// TIA Portal V20 export
// export: Created 2025-12-01T14:57:27.5166691Z, ExportSetting None, DisplayName Totally Integrated Automation Portal, DisplayVersion V20 Update 3, DisplayName TIA Portal Openness, DisplayVersion V20 Update 3, DisplayName TIA Portal Version Control Interface, DisplayVersion V20 Update 3, DisplayName STEP 7 Professional, DisplayVersion V20 Update 3, DisplayName STEP 7 Safety, DisplayVersion V20 Update 2, DisplayName WinCC Basic/Comfort/Advanced, DisplayVersion V20 Update 3, DisplayName WinCC Professional, DisplayVersion V20 Update 3, DisplayName WinCC Unified, DisplayVersion V20 Update 3
FUNCTION_BLOCK "FB606_SalidaMovil_Lateral_EnDesCarga_Quimarox"   // FB606, LAD
{ S7_Optimized_Access := 'FALSE' }
// stored: AutoNumber false, SetENOAutomatically false
   VAR_INPUT
      MesaSiguiente : UInt;
      MesaDeDescarga : UInt;
      ID_Quimarox : UInt;
      ID_Elemento : UInt;
      DestinoAsociado : UInt;
      EnTension : Bool;
      Termico : Bool;
      pHs_PosicionDescarga : Bool;
      pHs_Protrusion : Bool;
      En_PosicionDescarga : Bool;
      En_PosicionReposo : Bool;
      NXT_PTF : Bool;
      NXT_FTF : Bool;
      V_FILTRO_pHsPresencia : Int;
      Pto_Ajuste_1 : Int;   // en mm (paso a lenta en posicionamiento a descarga de transportador)
      Pto_Ajuste_2 : Int;   // en mm (timeout movimiento posicion descarga del transportador)
      Pto_Ajuste_3 : Int;   // en mm (paso a lenta en el proceso de descarga del peine)
      Pto_Ajuste_4 : Int;   // en mm (error protusion en descarga del elevador)
      Pto_Ajuste_5 : Int;   // en mm (paso a lenta en posicionamiento reposo del transportador)
      Pto_Ajuste_6 : Int;   // en mm (timeout movimiento posicion reposo del transportador)
   END_VAR
   VAR_OUTPUT
      NXT_DescargaActiva : Bool;
      NXT_AVTF : Bool;
      ElevadorEnLenta : Bool;
      PararElevador : Bool;
      Avance_SalidaMovil : Bool;
      Ir_PosicionReposo : Bool;
      Ir_PosicionDescarga : Bool;
   END_VAR
   VAR
      TMP_EnTension { S7_SetPoint := 'True'} : "FB910_CNT_UHS";
      FILTRO_pHsPresencia { S7_SetPoint := 'True'} : "FB910_CNT_UHS";
      EstadoAsociadoEnMesa : UInt;
      Ultimo_PeineTratado : UInt;
      Aux_PeineEnDesCarga { ExternalAccessible := 'False'; ExternalVisible := 'False'; ExternalWritable := 'False'} : UInt;
      Siguiente_ParaNosotros : Bool;
      PresenciaEnReset : Bool;
   END_VAR
   VAR_TEMP
      MesaQuimarox : UInt;
      NumeroUT : UInt;
      VagonSiguiente : UInt;
      EsMesaTL : Bool;
      FILTRO_PosicionDesCarga : Bool;
   END_VAR
BEGIN

NETWORK
TITLE = ERROR - Rearme
/////////////////////////////////////////////////////////////
/////////////////////////////////////////////////////////////
/////////////////////////////////////////////////////////////
// Rearne de Errores
      SET;
      A     "DB902_Estado_ZonaMesa".EstadoMesas[#MesaDeDescarga].Rearme_CBx;
      O     "DB902_Estado_ZonaMesa".EstadoMesas[#MesaDeDescarga].PerReset_CBx;
      R     "DB900_Estado_Mesas".EstadoVI[#MesaDeDescarga].Error_Mx;
      R     "DB900_Estado_Mesas".EstadoVI[#MesaDeDescarga].Err_Protusion;
      R     "DB900_Estado_Mesas".EstadoVI[#MesaDeDescarga].Err_Tout_Sacar;
      R     "DB900_Estado_Mesas".EstadoVI[#MesaDeDescarga].Err_Tout_Recoger;
      R     "DB900_Estado_Mesas".EstadoVI[#MesaDeDescarga].Err_DatosPLC;
      R     "DB900_Estado_Mesas".EstadoVI[#MesaDeDescarga].Err_Termico_E1_E3;
      R     "DB900_Estado_Mesas".EstadoVI[#MesaDeDescarga].Err_Perdida_PHs;



NETWORK
TITLE = RECEP OK DE LA ORDEN -- NO SE UTILIZA
/////////////////////////////////////////////////////////////
/////////////////////////////////////////////////////////////
/////////////////////////////////////////////////////////////
// RECEP OK DE LA ORDEN
      SET;
      AN    "DB841_Recepcion".Mesa[#MesaDeDescarga].Protocolo.Ord_S00;
      AN    "DB841_Recepcion".Mesa[#MesaDeDescarga].Protocolo.Ord_S01;
      AN    "DB841_Recepcion".Mesa[#MesaDeDescarga].Protocolo.Ord_S02;
      AN    "DB841_Recepcion".Mesa[#MesaDeDescarga].Protocolo.Ord_S03;
      NOT;
      =     "DB840_Emision".Mesa[#MesaDeDescarga].Protocolo.RecepOK;



NETWORK
TITLE = HMI - Manual
/////////////////////////////////////////////////////////////
/////////////////////////////////////////////////////////////
/////////////////////////////////////////////////////////////
// Para HMI >>> Manual
      SET;
      O     "DB902_Estado_ZonaMesa".EstadoMesas[#MesaDeDescarga].Manual_CBx;
      =     "DB900_Estado_Mesas".EstadoVI[#MesaDeDescarga].Manual;



NETWORK
TITLE = HMI - Entradas y Salidas de la Mesa
/////////////////////////////////////////////////////////////
/////////////////////////////////////////////////////////////
/////////////////////////////////////////////////////////////
// Entradas
      SET;
      A     #pHs_PosicionDescarga;
      =     "DB900_Estado_Mesas".EstadoVI[#MesaDeDescarga].En_PHS_1;
      SET;
      A     #pHs_Protrusion;
      =     "DB900_Estado_Mesas".EstadoVI[#MesaDeDescarga].En_pHs_Prot1;

      SET;
      A     #Termico;
      =     "DB900_Estado_Mesas".EstadoVI[#MesaDeDescarga].En_Termico1;


// Salidas
      SET;
      A     #Avance_SalidaMovil;
      =     "DB900_Estado_Mesas".EstadoVI[#MesaDeDescarga].Sa_Rod_Avance;
      SET;
      A     #Ir_PosicionReposo;
      =     "DB900_Estado_Mesas".EstadoVI[#MesaDeDescarga].Sa_Trans_Baj;
      SET;
      A     #Ir_PosicionDescarga;
      =     "DB900_Estado_Mesas".EstadoVI[#MesaDeDescarga].Sa_Trans_Sub;



NETWORK
TITLE = Comprobacion de que la MESA es de TRACKING
/////////////////////////////////////////////////////////////////////////////////////
/////////////////////////////////////////////////////////////////////////////////////
/////////////////////////////////////////////////////////////////////////////////////
// Comprobar si es una Mesa de Tracking o Routing
      SET;
      A     "DB850_DefinicionMesas".Mesa[#MesaDeDescarga].ConfigMesa.MesaTL;
      =     #EsMesaTL;



REGION Network 6: TMP - Espera En Tension
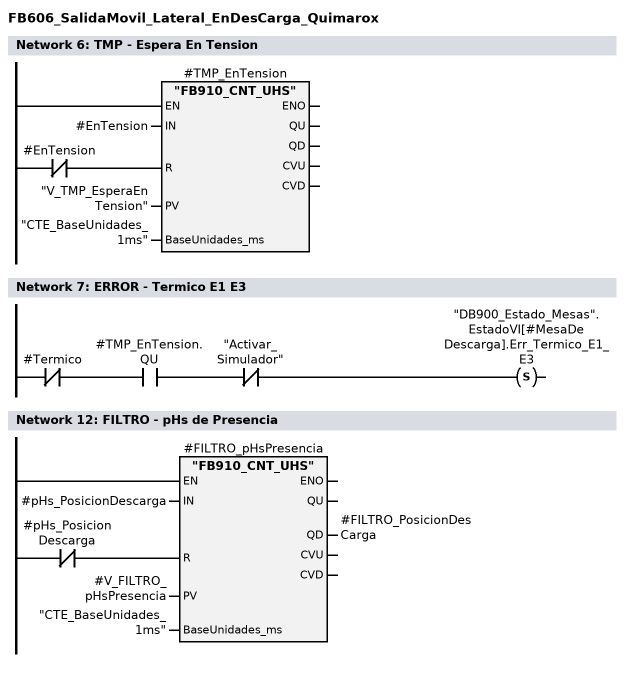
   RUNG wire#powerrail
      #TMP_EnTension(R := wire#w1, IN := #EnTension, PV := "V_TMP_EsperaEnTension", BaseUnidades_ms := "CTE_BaseUnidades_1ms", QU =>, QD =>, CVU =>, CVD =>)
   END_RUNG
   RUNG wire#powerrail
      I_Contact( #EnTension )
   END_RUNG wire#w1
   // the same network as SCL:
   #TMP_EnTension(IN := #EnTension,   // "FB910_CNT_UHS"
                  R := NOT #EnTension,
                  PV := "V_TMP_EsperaEnTension",
                  BaseUnidades_ms := "CTE_BaseUnidades_1ms");
END_REGION

REGION Network 7: ERROR - Termico E1 E3
   RUNG wire#powerrail
      I_Contact( #Termico )
      Contact( #TMP_EnTension.QU )
      I_Contact( "Activar_Simulador" )
      S_Coil( "DB900_Estado_Mesas".EstadoVI[#MesaDeDescarga].Err_Termico_E1_E3 )
   END_RUNG
   // the same network as SCL:
   IF NOT #Termico AND #TMP_EnTension.QU AND NOT "Activar_Simulador" THEN
       "DB900_Estado_Mesas".EstadoVI[#MesaDeDescarga].Err_Termico_E1_E3 := TRUE;
   END_IF;
END_REGION

NETWORK
TITLE = INICIALIZACION Previa
/////////////////////////////////////////////////////////////////////////////////////
/////////////////////////////////////////////////////////////////////////////////////
/////////////////////////////////////////////////////////////////////////////////////
      CLR;
      =     #ElevadorEnLenta;
      =     #PararElevador;

      CLR;
      =     #NXT_DescargaActiva;
      =     #NXT_AVTF;

      CLR;
      =     #Avance_SalidaMovil;
      =     #Ir_PosicionReposo;
      =     #Ir_PosicionDescarga;



NETWORK
TITLE = SISTEMA - Paro Blando
/////////////////////////////////////////////////////////////
/////////////////////////////////////////////////////////////
/////////////////////////////////////////////////////////////
// - Inicializar Variables de PARO BLANDO
      CLR;
      =     "DB900_Estado_Mesas".EstadoVI[#MesaDeDescarga].Paro_Blando;

/////////////////////////////////////////////////////////////
// - Existe PARO BLANDO ???
      SET;
      AN    "DB902_Estado_ZonaMesa".EstadoMesas[#MesaDeDescarga].ParoBlando_CBx;
      JC    NoRealizandose_ParoBlando;

/////////////////////////////////////////////////////////////
// - Fin de PARO BLANDO
      SET;
      =     "DB900_Estado_Mesas".EstadoVI[#MesaDeDescarga].Paro_Blando;


/////////////////////////////////////////////////////////////
/////////////////////////////////////////////////////////////
/////////////////////////////////////////////////////////////
// - Final Tratamiento del PARO BLANDO
NoRealizandose_ParoBlando:NOP   0;



NETWORK
TITLE = SISTEMA - Reset
/////////////////////////////////////////////////////////////
/////////////////////////////////////////////////////////////
/////////////////////////////////////////////////////////////
// -- Inicializar Variables de RESET
      SET;
      AN    "DB902_Estado_ZonaMesa".EstadoMesas[#MesaDeDescarga].PerReset_CBx;
      R     "DB900_Estado_Mesas".EstadoVI[#MesaDeDescarga].Fin_VI;
      R     #PresenciaEnReset;

/////////////////////////////////////////////////////////////
/////////////////////////////////////////////////////////////
/////////////////////////////////////////////////////////////
// - Existe RESET ??
      SET;
      AN    "DB902_Estado_ZonaMesa".EstadoMesas[#MesaDeDescarga].PerReset_CBx;
      JC    NoRealizandose_Reset;

      L     0;  // Estado de La Mesa = 0
      T     #EstadoAsociadoEnMesa;
      T     #Ultimo_PeineTratado;

      SET;
      =     "DB900_Estado_Mesas".EstadoVI[#MesaDeDescarga].Etapas_Reset;

/////////////////////////////////////////////////////////////
/////////////////////////////////////////////////////////////
/////////////////////////////////////////////////////////////
// - Emision de Presencia en caso de Reset
      SET;  // Presencia >>> Reset Total
      A     #pHs_PosicionDescarga;
      A     "DB831_Mesas".Mesas[#MesaDeDescarga].Memorias.M_ResetTotal;
      AN    #PresenciaEnReset;
      JC    Enviar_PresenciaEnResetTotal;

      SET;  // Presencia >>> Reset Parcial
      A     #pHs_PosicionDescarga;
      A     "DB831_Mesas".Mesas[#MesaDeDescarga].Memorias.M_ResetParcial;
      AN    #PresenciaEnReset;
      JC    Enviar_PresenciaEnResetParcial;

      JU    Final_PresenciaEnReset;

// - Presencia en Reset TOTAL >>> Enviar NUUT
Enviar_PresenciaEnResetTotal:NOP   0;
      CALL  "FC723_InsertarUT_EnMesa"
      ( MesaActual := #MesaDeDescarga,
        NumeroUT   := #NumeroUT
      );
      L     132;  // Envio de Nueva UT en RESET
      T     "DB812_UTs_Control".UT[#NumeroUT].EstadoEventoAGenerar;

      SET;  // Ya esta Avisado el JdT
      S     #PresenciaEnReset;

      JU    Final_PresenciaEnReset;

// - Presencia en Reset Parcial >>> Enviar LOCA en Reset Pantalla
Enviar_PresenciaEnResetParcial:NOP   0;
      L     "DB810_ColasMesas".Colas[#MesaDeDescarga].UT_PrimeraMesa;
      T     #NumeroUT;

      L     #NumeroUT;  // Comprobar que Existe UT
      L     0;
      ==I;
      JC    ErrorDatosCargada;

      L     101;  // Envio de LOCA en RESET
      T     "DB812_UTs_Control".UT[#NumeroUT].EstadoEventoAGenerar;

      SET;  // Ya esta Avisado el JdT
      S     #PresenciaEnReset;

      JU    Final_PresenciaEnReset;

// - Final de la Presencia En Reset
Final_PresenciaEnReset:NOP   0;


/////////////////////////////////////////////////////////////
/////////////////////////////////////////////////////////////
/////////////////////////////////////////////////////////////
// - Fin de RESET
      SET;  // Con Presencia de Carga >>> TOTAL
      A(;
      L     "DB810_ColasMesas".Colas[#MesaDeDescarga].UT_PrimeraMesa;
      L     0;
      ==I;
      );
      A     #pHs_PosicionDescarga;
      A     #PresenciaEnReset;
      A     "DB831_Mesas".Mesas[#MesaDeDescarga].Memorias.M_ResetTotal;
      S     "DB900_Estado_Mesas".EstadoVI[#MesaDeDescarga].Fin_VI;

      SET;  // Con Presencia de Carga >>> PARCIAL
      A     #pHs_PosicionDescarga;
      A     #PresenciaEnReset;
      A     "DB831_Mesas".Mesas[#MesaDeDescarga].Memorias.M_ResetParcial;
      S     "DB900_Estado_Mesas".EstadoVI[#MesaDeDescarga].Fin_VI;


      SET;  // Sin Presencia de Carga
      AN    #pHs_PosicionDescarga;
      S     "DB900_Estado_Mesas".EstadoVI[#MesaDeDescarga].Fin_VI;

      BE;

/////////////////////////////////////////////////////////////
/////////////////////////////////////////////////////////////
/////////////////////////////////////////////////////////////
// - Final Tratamiento del RESET
NoRealizandose_Reset:NOP   0;



NETWORK
TITLE = >>>>>>>>>>>>>>>>>>>>>>>>>>>>>>>>>>>>>>>>>>>>>>>>>>>>>>>>>>>>>>>>>>>

REGION Network 12: FILTRO - pHs de Presencia
   RUNG wire#powerrail
      #FILTRO_pHsPresencia(R := wire#w1, IN := #pHs_PosicionDescarga, PV := #V_FILTRO_pHsPresencia, BaseUnidades_ms := "CTE_BaseUnidades_1ms", QU =>, QD => #FILTRO_PosicionDesCarga, CVU =>, CVD =>)
   END_RUNG
   RUNG wire#powerrail
      I_Contact( #pHs_PosicionDescarga )
   END_RUNG wire#w1
   // the same network as SCL:
   #FILTRO_pHsPresencia(IN := #pHs_PosicionDescarga,   // "FB910_CNT_UHS"
                        R := NOT #pHs_PosicionDescarga,
                        PV := #V_FILTRO_pHsPresencia,
                        BaseUnidades_ms := "CTE_BaseUnidades_1ms",
                        QD => #FILTRO_PosicionDesCarga);
END_REGION

NETWORK
TITLE = >>>>>>>>>>>>>>>>>>>>>>>>>>>>>>>>>>>>>>>>>>>>>>>>>>>>>>>>>>>>>>>>>>>

NETWORK
TITLE = DISTRIBUCION >>> Control Etapa Activa
/////////////////////////////////////////////////////////////////////////////////////
/////////////////////////////////////////////////////////////////////////////////////
/////////////////////////////////////////////////////////////////////////////////////
// listado de saltos de programa
      L     #EstadoAsociadoEnMesa;
      JL    ETAPA_PorDefecto;

      JU    ETAPA_00_EnReset;
      JU    ETAPA_01_EnReposo;

      JU    ETAPA_02_MoverPosicionDescarga;
      JU    ETAPA_03_PreparadaDescarga;
      JU    ETAPA_04_EnEsperaDescarga;
      JU    ETAPA_05_EnDescargaActiva;
      JU    ETAPA_06_FinDescarga;
      JU    ETAPA_07_MoverPosicionReposo;

      JU    ETAPA_PorDefecto;
      JU    ETAPA_PorDefecto;

      JU    ETAPA_10_ResetVacio_MoverPosicionDeReposo;
      JU    ETAPA_11_ResetCargado_EnEsperaDesCarga;
      JU    ETAPA_12_ResetCargado_EnDescargaActiva;
      JU    ETAPA_13_ResetCargado_FinDescarga;
      JU    ETAPA_14_ResetCargado_MoverPosicionReposo;

ETAPA_PorDefecto:JU    FinFuncion;



NETWORK
TITLE = ETAPA 00 >>> En Reset
/////////////////////////////////////////////////////////////////////////////////////
/////////////////////////////////////////////////////////////////////////////////////
/////////////////////////////////////////////////////////////////////////////////////
ETAPA_00_EnReset:NOP   0;
      SET;
      =     "DB900_Estado_Mesas".EstadoVI[#MesaDeDescarga].Etapas_Reset;


/////////////////////////////////////////////////////////////////////////////////////
// error de protusion
      SET;
      AN    #pHs_Protrusion;
      JC    ErrorProtrusion;

/////////////////////////////////////////////////////////////////////////////////////
// Tiene que estar en Marcha y Sin Error para continuar
      SET;
      AN    "DB902_Estado_ZonaMesa".EstadoMesas[#MesaDeDescarga].Marcha_CBx;
      O     "DB902_Estado_ZonaMesa".EstadoMesas[#MesaDeDescarga].Error_CBx;
      JC    ET00_PararElevador;


/////////////////////////////////////////////////////////////////////////////////////
/////////////////////////////////////////////////////////////////////////////////////
//  Vacio >>> No esta en Reposo
      SET;
      AN    #FILTRO_PosicionDesCarga;
      AN    #En_PosicionReposo;
      JC    ET00_IrEtapa_10_ResetVacio_MoverPosicionReposo;

//  Vacio >>> Esta en Reposo
      SET;
      AN    #FILTRO_PosicionDesCarga;
      A     #En_PosicionReposo;
      JC    ET00_IrEtapa_01_EnReposo;


/////////////////////////////////////////////////////////////////////////////////////
/////////////////////////////////////////////////////////////////////////////////////
//  Lleno >>> No Esta en Reposo
      SET;
      A     #FILTRO_PosicionDesCarga;
      AN    #En_PosicionReposo;
      JC    ET00_IrEtapa_11_ResetCargado_EnEsperaDesCarga;

//  Lleno >>> Esta en Reposo
      SET;
      A     #FILTRO_PosicionDesCarga;
      A     #En_PosicionReposo;
      JC    ErrorMoverPosicionReposo;

      BE;


/////////////////////////////////////////////////////////////////////////////////////
/////////////////////////////////////////////////////////////////////////////////////
/////////////////////////////////////////////////////////////////////////////////////
ET00_PararElevador:NOP   0;
      SET;
      =     #PararElevador;
      BE;


/////////////////////////////////////////////////////////////////////////////////////
/////////////////////////////////////////////////////////////////////////////////////
/////////////////////////////////////////////////////////////////////////////////////
ET00_IrEtapa_01_EnReposo:NOP   0;
      L     1;
      T     #EstadoAsociadoEnMesa;
      JU    ETAPA_01_EnReposo;

/////////////////////////////////////////////////////////////////////////////////////
ET00_IrEtapa_10_ResetVacio_MoverPosicionReposo:NOP   0;
      L     10;
      T     #EstadoAsociadoEnMesa;
      JU    ETAPA_10_ResetVacio_MoverPosicionDeReposo;

/////////////////////////////////////////////////////////////////////////////////////
ET00_IrEtapa_11_ResetCargado_EnEsperaDesCarga:NOP   0;
      SET;  // No existe UT >>> Error de Datos
      A(;
      L     "DB810_ColasMesas".Colas[#MesaDeDescarga].UT_PrimeraMesa;
      L     0;
      ==I;
      );
      AN    #EsMesaTL;
      JC    ErrorDatosCargada;

      L     11;
      T     #EstadoAsociadoEnMesa;
      JU    ETAPA_11_ResetCargado_EnEsperaDesCarga;



NETWORK
TITLE = ETAPA 01 >>> En Reposo
/////////////////////////////////////////////////////////////////////////////////////
/////////////////////////////////////////////////////////////////////////////////////
/////////////////////////////////////////////////////////////////////////////////////
// Estado de reposo esperando a que llegue una carga para este destino
ETAPA_01_EnReposo:NOP   0;
      SET;
      =     "DB900_Estado_Mesas".EstadoVI[#MesaDeDescarga].Etapa_Vacia;


/////////////////////////////////////////////////////////////////////////////////////
// miramos si ya hemos comprobado el peine que está delante nuestro
      SET;
      L     "DB602_ElementosQuimarox".Quimarox[#ID_Quimarox].Elementos[#ID_Elemento].Numero_carrier;
      L     #Ultimo_PeineTratado;
      ==I;
      JC    ET01_SinPeineEnVentana;

/////////////////////////////////////////////////////////////////////////////////////
// si no hemos comprobado el peine, comprobamos si tenemos un peine en ventana
      SET;
      AN    "DB602_ElementosQuimarox".Quimarox[#ID_Quimarox].Elementos[#ID_Elemento].Hay_Carrier_en_ventana;
      JC    ET01_SinPeineEnVentana;

/////////////////////////////////////////////////////////////////////////////////////
// si no ha saltado es porque el carrier está en ventana. Comprobamos si es para nosotros
      SET;
      L     "DB602_ElementosQuimarox".Quimarox[#ID_Quimarox].Elementos[#ID_Elemento].Numero_carrier;
      T     #Aux_PeineEnDesCarga;

      SET;
      L     "DB601_PeinesQuimarox".Quimarox[#ID_Quimarox].vagon[#Aux_PeineEnDesCarga].Destino_principal;
      L     #DestinoAsociado;
      ==I;
      JC    ET01_PeineParaLaMesa;

/////////////////////////////////////////////////////////////////////////////////////
// si no es para mi, me guardo que he chequeado el peine para no volver a comprobarlo
      L     "DB602_ElementosQuimarox".Quimarox[#ID_Quimarox].Elementos[#ID_Elemento].Numero_carrier;
      T     #Ultimo_PeineTratado;
      BE;


/////////////////////////////////////////////////////////////////////////////////////
/////////////////////////////////////////////////////////////////////////////////////
/////////////////////////////////////////////////////////////////////////////////////
ET01_SinPeineEnVentana:NOP   0;
      SET;  // Esta TOTALMENTE libre ?
      A(;
      O     #FILTRO_PosicionDesCarga;
      ON    #pHs_Protrusion;
      );
      JCN   FinFuncion;
      JU    ErrorProtrusion;


/////////////////////////////////////////////////////////////////////////////////////
/////////////////////////////////////////////////////////////////////////////////////
/////////////////////////////////////////////////////////////////////////////////////
ET01_PeineParaLaMesa:NOP   0;
      L     2;
      T     #EstadoAsociadoEnMesa;
      L     "DB602_ElementosQuimarox".Quimarox[#ID_Quimarox].Elementos[#ID_Elemento].Numero_carrier;
      T     #Ultimo_PeineTratado;

      JU    ETAPA_02_MoverPosicionDescarga;



NETWORK
TITLE = ETAPA 02 >>> Mover a Posicion de Descarga
/////////////////////////////////////////////////////////////////////////////////////
/////////////////////////////////////////////////////////////////////////////////////
/////////////////////////////////////////////////////////////////////////////////////
// inicio del proceso de descarga
// antes de iniciar la descarga tenemos que colocar el transportador en la posicion de descarga
ETAPA_02_MoverPosicionDescarga:NOP   0;
      SET;
      =     "DB900_Estado_Mesas".EstadoVI[#MesaDeDescarga].Etapas_Carga_E0;


/////////////////////////////////////////////////////////////////////////////////////
      SET;
      A     #En_PosicionDescarga;
      JC    ET02_IrEtapa_03_PreparadoParaDesCarga;

/////////////////////////////////////////////////////////////////////////////////////
      SET;
      =     #Ir_PosicionDescarga;
      CLR;
      =     #Ir_PosicionReposo;

/////////////////////////////////////////////////////////////////////////////////////
// como estamos metiendo el transportador, tenemos que vigilar que no tarda demasiado en entrar
      L     "DB602_ElementosQuimarox".Quimarox[#ID_Quimarox].Elementos[#ID_Elemento].Avance_carrier;  // #datos_elemento.Avance_carrier
      L     #Pto_Ajuste_1;
      <=I;
      JC    ET02_VelocidadNormal;

      SET;
      =     #ElevadorEnLenta;

      L     "DB602_ElementosQuimarox".Quimarox[#ID_Quimarox].Elementos[#ID_Elemento].Avance_carrier;  //#datos_elemento.Avance_carrier
      L     #Pto_Ajuste_2;
      >=I;
      JC    ErrorMoverPosicionDescarga;  // error de movimiento al sacar el transportador

      BE;


/////////////////////////////////////////////////////////////////////////////////////
ET02_VelocidadNormal:CLR;
      =     #ElevadorEnLenta;
      BE;

/////////////////////////////////////////////////////////////////////////////////////
ET02_IrEtapa_03_PreparadoParaDesCarga:CLR;
      =     #Ir_PosicionDescarga;
      L     3;
      T     #EstadoAsociadoEnMesa;

      JU    ETAPA_03_PreparadaDescarga;



NETWORK
TITLE = ETAPA 03 >>> Etapa Preparado para el Proceso de Descarga
/////////////////////////////////////////////////////////////////////////////////////
/////////////////////////////////////////////////////////////////////////////////////
/////////////////////////////////////////////////////////////////////////////////////
// espera a la descarga activa
// antes de iniciar la descarga tenemos que esperar a ver el detector de la descarga
ETAPA_03_PreparadaDescarga:NOP   0;
      SET;
      =     "DB900_Estado_Mesas".EstadoVI[#MesaDeDescarga].Etapas_Carga_E0;


/////////////////////////////////////////////////////////////////////////////////////
      SET;
      A     #FILTRO_PosicionDesCarga;
      JC    ET03_IrEtapa_04_EnEsPeraDesCarga;


/////////////////////////////////////////////////////////////////////////////////////
// tenemos que comprobar si seguimos en la ventana, sino nos retiramos
      SET;
      AN    #pHs_Protrusion;
      JC    ErrorProtrusion;

/////////////////////////////////////////////////////////////////////////////////////
      SET;
      A     "DB602_ElementosQuimarox".Quimarox[#ID_Quimarox].Elementos[#ID_Elemento].Hay_Carrier_en_ventana;  //#datos_elemento.Hay_Carrier_en_ventana
      JC    FinFuncion;

/////////////////////////////////////////////////////////////////////////////////////
      SET;
      AN    "DB602_ElementosQuimarox".Quimarox[#ID_Quimarox].Elementos[#ID_Elemento].Hay_Carrier_en_ventana;  // #datos_elemento.Hay_Carrier_en_ventana
      A     #Siguiente_ParaNosotros;
      JC    FinFuncion;


/////////////////////////////////////////////////////////////////////////////////////
// nieves: la siguiente condicion creo que no está bien, no tiene sentido ir a la et6
      SET;
      A     "DB602_ElementosQuimarox".Quimarox[#ID_Quimarox].Elementos[#ID_Elemento].Hay_Carrier_en_ventana;  // #datos_elemento.Hay_Carrier_en_ventana
      A     #Siguiente_ParaNosotros;
      JC    ET03_IrEtapa_07_MoverPosicionReposo;

      BE;


/////////////////////////////////////////////////////////////////////////////////////
ET03_IrEtapa_07_MoverPosicionReposo:NOP   0;
      L     7;
      T     #EstadoAsociadoEnMesa;
      JU    ETAPA_07_MoverPosicionReposo;

/////////////////////////////////////////////////////////////////////////////////////
// si hemos visto el detector, es que nos tenemos que poner en el estado de descarga activa.
ET03_IrEtapa_04_EnEsPeraDesCarga:NOP   0;
      L     "DB602_ElementosQuimarox".Quimarox[#ID_Quimarox].Elementos[#ID_Elemento].Numero_carrier;
      T     #Aux_PeineEnDesCarga;

// Emision del Evento del Quimarox
      L     "CTE_Evento_QDES";
      T     "DB601_PeinesQuimarox".Quimarox[#ID_Quimarox].vagon[#Aux_PeineEnDesCarga].EventoAGenerar;
      L     #MesaDeDescarga;
      L     "CTE_OffsetMesa";
      +I;
      T     "DB601_PeinesQuimarox".Quimarox[#ID_Quimarox].vagon[#Aux_PeineEnDesCarga].Mesa_descarga;

/////////////////////////////////////////////////////////////////////////////////////
/////////////////////////////////////////////////////////////////////////////////////
/////////////////////////////////////////////////////////////////////////////////////
// Comprobar Tipo de Mesa
      SET;
      A     #EsMesaTL;
      JC    ET03_Final_RecogerDatosDelPeine;

/////////////////////////////////////////////////////////////////////////////////////
// TRACKING - INICIO - Recoger Datos del Peine
      SET;
      L     "DB601_PeinesQuimarox".Quimarox[#ID_Quimarox].vagon[#Aux_PeineEnDesCarga].DatosCarga.Mckey;
      L     0;
      ==D;
      JC    ET03_TRACKING_CrearNueva_UT;
      JU    ET03_TRACKING_Crear_UT;


/////////////////////////////////////////////////////////////////////////////////////
// TRAKING - NuevaUT en la Mesa
ET03_TRACKING_Crear_UT:NOP   0;
      CALL  "FC721_CrearUT_EnMesa"
      ( McKey      := "DB601_PeinesQuimarox".Quimarox[#ID_Quimarox].vagon[#Aux_PeineEnDesCarga].DatosCarga.Mckey,
        MesaActual := #MesaDeDescarga,
        NumeroUT   := #NumeroUT
      );

      L     100;  // Emitir evento LOCA
      T     "DB812_UTs_Control".UT[#NumeroUT].EstadoEventoAGenerar;

      L     "DB601_PeinesQuimarox".Quimarox[#ID_Quimarox].vagon[#Aux_PeineEnDesCarga].DatosCarga.MesaDestino;
      T     "DB812_UTs_Control".UT[#NumeroUT].MesaDestino;
      T     "DB812_UTs_Control".UT[#NumeroUT].MesaIntermedia;
      T     "DB813_UTs_Ruta".UT[#NumeroUT].Ruta[0];

      JU    ET03_Final_RecogerDatosDelPeine;


/////////////////////////////////////////////////////////////////////////////////////
// TRAKING - NuevaUT en la Mesa
ET03_TRACKING_CrearNueva_UT:NOP   0;
      JU    ET03_Final_RecogerDatosDelPeine;


/////////////////////////////////////////////////////////////////////////////////////
// Final de la Recogida de Datos del Peine
ET03_Final_RecogerDatosDelPeine:NOP   0;
      L     4;
      T     #EstadoAsociadoEnMesa;
      JU    ETAPA_04_EnEsperaDescarga;



NETWORK
TITLE = ETAPA 04 >>> Inicio de Descarga
/////////////////////////////////////////////////////////////////////////////////////
/////////////////////////////////////////////////////////////////////////////////////
/////////////////////////////////////////////////////////////////////////////////////
// Proceso de descarga activa
// Tenemos que esperar a dejar de ver los dos detectores antes de dar por finalizado el proceso de descarga
ETAPA_04_EnEsperaDescarga:NOP   0;
      SET;
      =     "DB900_Estado_Mesas".EstadoVI[#MesaDeDescarga].Etapa_Cargada;


/////////////////////////////////////////////////////////////////////////////////////
      SET;
      =     #NXT_AVTF;

      SET;
      A     #NXT_PTF;
      JC    ET04_IrEtapa_05_EnDesCargaActiva;

/////////////////////////////////////////////////////////////////////////////////////
// tenemos que comprobar si seguimos en la ventana, sino nos retiramos
      SET;
      AN    #pHs_Protrusion;
      JC    ErrorProtrusion;

/////////////////////////////////////////////////////////////////////////////////////
// nieves. aqui hay que vigilar la ventana del peine para ver si entramos en una zona peligrosa.
// añadir luego control de la ventana de descarga
      SET;
      L     "DB602_ElementosQuimarox".Quimarox[#ID_Quimarox].Elementos[#ID_Elemento].Avance_carrier;  //#datos_elemento.Avance_carrier
      L     #Pto_Ajuste_3;
      <=I;
      JC    FinFuncion;

      SET;
      =     #ElevadorEnLenta;

/////////////////////////////////////////////////////////////////////////////////////
      SET;
      AN    "DB602_ElementosQuimarox".Quimarox[#ID_Quimarox].Elementos[#ID_Elemento].Hay_Carrier_en_ventana;  // #datos_elemento.Hay_Carrier_en_ventana
      A(;
      ON    #pHs_Protrusion;
      O     #FILTRO_PosicionDesCarga;
      );
      JC    ET04_PararElevador;

/////////////////////////////////////////////////////////////////////////////////////
      SET;
      A     "DB602_ElementosQuimarox".Quimarox[#ID_Quimarox].Elementos[#ID_Elemento].Hay_Carrier_en_ventana;  // #datos_elemento.Hay_Carrier_en_ventana
      A(;
      L     "DB602_ElementosQuimarox".Quimarox[#ID_Quimarox].Elementos[#ID_Elemento].Avance_carrier;  // #datos_elemento.Avance_carrier
      L     #Pto_Ajuste_4;
      >=I;
      );
      ON    #pHs_Protrusion;
      O     #FILTRO_PosicionDesCarga;
      JCN   FinFuncion;

      JU    ET04_PararElevador;

/////////////////////////////////////////////////////////////////////////////////////
ET04_PararElevador:NOP   0;
      SET;
      =     #PararElevador;
      BE;

/////////////////////////////////////////////////////////////////////////////////////
ET04_IrEtapa_05_EnDesCargaActiva:NOP   0;
      L     5;
      T     #EstadoAsociadoEnMesa;
      JU    ETAPA_05_EnDescargaActiva;



NETWORK
TITLE = ETAPA 05 >>> Descarga Activa
/////////////////////////////////////////////////////////////////////////////////////
/////////////////////////////////////////////////////////////////////////////////////
/////////////////////////////////////////////////////////////////////////////////////
// Proceso de descarga activa
// Tenemos que esperar a dejar de ver los dos detectores antes de dar por finalizado el proceso de descarga
ETAPA_05_EnDescargaActiva:NOP   0;
      SET;
      =     "DB900_Estado_Mesas".EstadoVI[#MesaDeDescarga].Etapas_Descarga_S3;


/////////////////////////////////////////////////////////////////////////////////////

      SET;
      =     #NXT_AVTF;
      =     #NXT_DescargaActiva;

      SET;
      A     #NXT_PTF;
      =     #Avance_SalidaMovil;

      SET;
      AN    #FILTRO_PosicionDesCarga;
      A     #pHs_Protrusion;
      A     #NXT_FTF;
      JC    ET05_IrEtapa_06_FinDescarga;


/////////////////////////////////////////////////////////////////////////////////////
// nieves. aqui hay que vigilar la ventana del peine para ver si entramos en una zona peligrosa.
// añadir luego control de la ventana de descarga
      SET;
      L     "DB602_ElementosQuimarox".Quimarox[#ID_Quimarox].Elementos[#ID_Elemento].Avance_carrier;  //#datos_elemento.Avance_carrier
      L     #Pto_Ajuste_3;
      <=I;
      JC    FinFuncion;

      SET;
      =     #ElevadorEnLenta;

/////////////////////////////////////////////////////////////////////////////////////
      SET;
      AN    "DB602_ElementosQuimarox".Quimarox[#ID_Quimarox].Elementos[#ID_Elemento].Hay_Carrier_en_ventana;  // #datos_elemento.Hay_Carrier_en_ventana
      A(;
      ON    #pHs_Protrusion;
      O     #FILTRO_PosicionDesCarga;
      );
      JC    ET05_PararElevador;

/////////////////////////////////////////////////////////////////////////////////////
      SET;
      A     "DB602_ElementosQuimarox".Quimarox[#ID_Quimarox].Elementos[#ID_Elemento].Hay_Carrier_en_ventana;  // #datos_elemento.Hay_Carrier_en_ventana
      A(;
      L     "DB602_ElementosQuimarox".Quimarox[#ID_Quimarox].Elementos[#ID_Elemento].Avance_carrier;  // #datos_elemento.Avance_carrier
      L     #Pto_Ajuste_4;
      >=I;
      );
      ON    #pHs_Protrusion;
      O     #FILTRO_PosicionDesCarga;
      JCN   FinFuncion;

      JU    ET05_PararElevador;

/////////////////////////////////////////////////////////////////////////////////////
ET05_PararElevador:NOP   0;
      SET;
      =     #PararElevador;
      BE;

/////////////////////////////////////////////////////////////////////////////////////
ET05_IrEtapa_06_FinDescarga:NOP   0;
      CLR;
      =     #NXT_DescargaActiva;
      =     #NXT_AVTF;
      =     #ElevadorEnLenta;
      =     #PararElevador;
      =     #Avance_SalidaMovil;

      L     6;
      T     #EstadoAsociadoEnMesa;
      JU    ETAPA_06_FinDescarga;



NETWORK
TITLE = ETAPA 06 >>> Fin Descarga
/////////////////////////////////////////////////////////////////////////////////////
/////////////////////////////////////////////////////////////////////////////////////
/////////////////////////////////////////////////////////////////////////////////////
// antes de saltar al inicio proceso reposo, vamos a ver si el siguiente peine que va a llegar
// tiene también una carga para nosotros. Para eso tenemos que sacar el dato del peine siguiente.
ETAPA_06_FinDescarga:NOP   0;
      SET;
      =     "DB900_Estado_Mesas".EstadoVI[#MesaDeDescarga].Etapas_Descarga_S3;


/////////////////////////////////////////////////////////////////////////////////////
      CLR;
      =     #NXT_DescargaActiva;
      =     #NXT_AVTF;
      =     #ElevadorEnLenta;
      =     #PararElevador;
      =     #Avance_SalidaMovil;


/////////////////////////////////////////////////////////////////////////////////////
/////////////////////////////////////////////////////////////////////////////////////
/////////////////////////////////////////////////////////////////////////////////////
      JU    ET06_FINAL_PasoDeDatos;


/////////////////////////////////////////////////////////////////////////////////////
/////////////////////////////////////////////////////////////////////////////////////
/////////////////////////////////////////////////////////////////////////////////////
ET06_FINAL_PasoDeDatos:NOP   0;
      L     "DB602_ElementosQuimarox".Quimarox[#ID_Quimarox].Elementos[#ID_Elemento].Numero_carrier;
      L     1;
      +I;
      T     #VagonSiguiente;

/////////////////////////////////////////////////////////////////////////////////////
// antes de buscar en los datos del siguiente vagon, tenemos que ver si el número es coherente.
      SET;
      L     #VagonSiguiente;
      L     "DB600_ConfigQuimarox".Quimarox[#ID_Quimarox].datos_config.Numero_vagones;  //#DatosConfig.Numero_vagones// numero máximo de vagones que existen
      <=I;
      JC    ET06_Comprueba_SiguientePeine;

// si no ha saltado a busca, es que hemos superado el máximo
      L     1;
      T     #VagonSiguiente;

/////////////////////////////////////////////////////////////////////////////////////
// comprobamos si el peine está cargado, y si también es para nosotros no tenemos que pasar por la posicion de reposo
ET06_Comprueba_SiguientePeine:NOP   0;
      SET;
      A     "DB601_PeinesQuimarox".Quimarox[#ID_Quimarox].vagon[#VagonSiguiente].Carrier_Cargado;  //#datos_peine_tmp.Carrier_Cargado
      A(;
      L     "DB601_PeinesQuimarox".Quimarox[#ID_Quimarox].vagon[#VagonSiguiente].Destino_principal;
      L     #DestinoAsociado;
      ==I;
      );
      JC    ET06_IrEtapa_03_PreparadaDesCarga;
      JU    ET06_IrEtapa_07_MoverPosicionReposo;

/////////////////////////////////////////////////////////////////////////////////////
// si el vagón está cargado, y la carga es para nuestro destino, volvemos a la etapa 3, espera a la descarga
ET06_IrEtapa_03_PreparadaDesCarga:NOP   0;
      SET;
      =     #Siguiente_ParaNosotros;

      L     3;
      T     #EstadoAsociadoEnMesa;
      JU    ETAPA_03_PreparadaDescarga;

/////////////////////////////////////////////////////////////////////////////////////
// si no está cargado o no es para nosotros la carga, tenemos que volver a la posición de reposo.
ET06_IrEtapa_07_MoverPosicionReposo:NOP   0;
      CLR;
      =     #Siguiente_ParaNosotros;

      L     7;
      T     #EstadoAsociadoEnMesa;
      JU    ETAPA_07_MoverPosicionReposo;



NETWORK
TITLE = ETAPA 07 >>> Mover a Posicion de Reposo
/////////////////////////////////////////////////////////////////////////////////////
/////////////////////////////////////////////////////////////////////////////////////
/////////////////////////////////////////////////////////////////////////////////////
// inicio del proceso de vuelta a reposo
ETAPA_07_MoverPosicionReposo:NOP   0;
      SET;
      =     "DB900_Estado_Mesas".EstadoVI[#MesaDeDescarga].Etapas_Descarga_S3;


/////////////////////////////////////////////////////////////////////////////////////
      CLR;
      =     #NXT_AVTF;
      =     #NXT_DescargaActiva;
      =     #Avance_SalidaMovil;

      SET;
      A     #En_PosicionReposo;
      JC    ET07_REPOSO_IrEtapa_01_EnReposo;

/////////////////////////////////////////////////////////////////////////////////////
      SET;
      =     #Ir_PosicionReposo;

      L     "DB602_ElementosQuimarox".Quimarox[#ID_Quimarox].Elementos[#ID_Elemento].Avance_carrier;  //#datos_elemento.Avance_carrier
      L     #Pto_Ajuste_5;
      <=I;
      JC    ET07_REPOSO_VelocidadNormal;

      SET;
      =     #ElevadorEnLenta;

/////////////////////////////////////////////////////////////////////////////////////
      SET;
      L     "DB602_ElementosQuimarox".Quimarox[#ID_Quimarox].Elementos[#ID_Elemento].Avance_carrier;  // #datos_elemento.Avance_carrier
      L     #Pto_Ajuste_6;
      >=I;
      JC    ErrorMoverPosicionReposo;  // error de movimiento al meter el transportador

/////////////////////////////////////////////////////////////////////////////////////
      SET;
      AN    "DB602_ElementosQuimarox".Quimarox[#ID_Quimarox].Elementos[#ID_Elemento].Hay_Carrier_en_ventana;  //#datos_elemento.Hay_Carrier_en_ventana
      JC    ErrorMoverPosicionReposo;

      BE;

/////////////////////////////////////////////////////////////////////////////////////
ET07_REPOSO_VelocidadNormal:NOP   0;
      CLR;
      =     #ElevadorEnLenta;
      BE;

/////////////////////////////////////////////////////////////////////////////////////
ET07_REPOSO_IrEtapa_01_EnReposo:NOP   0;
      CLR;
      =     #Ir_PosicionReposo;
      =     #ElevadorEnLenta;

      L     1;
      T     #EstadoAsociadoEnMesa;
      BE;



NETWORK
TITLE = >>>>>>>>>>>>>>>>>>>>>>>>>>>>>>>>>>>>>>>>>>>>>>>>>>>>>>>>>>>>>>>>>>>

NETWORK
TITLE = ETAPA 10 >>> RESET VACIO >>> Mover Posicion de Reposo
/////////////////////////////////////////////////////////////////////////////////////
/////////////////////////////////////////////////////////////////////////////////////
/////////////////////////////////////////////////////////////////////////////////////
ETAPA_10_ResetVacio_MoverPosicionDeReposo:NOP   0;
      SET;
      =     "DB900_Estado_Mesas".EstadoVI[#MesaDeDescarga].Etapas_Reset;


/////////////////////////////////////////////////////////////////////////////////////
      SET;
      AN    #pHs_Protrusion;
      JC    ErrorProtrusion;


/////////////////////////////////////////////////////////////////////////////////////
/////////////////////////////////////////////////////////////////////////////////////
/////////////////////////////////////////////////////////////////////////////////////
      SET;
      A     #En_PosicionReposo;
      JC    ET10_IrEtapa_1_ResetVacio_EnReposo;


/////////////////////////////////////////////////////////////////////////////////////
      SET;
      =     #Ir_PosicionReposo;
      =     #PararElevador;

      CLR;
      =     #Ir_PosicionDescarga;

      BE;


/////////////////////////////////////////////////////////////////////////////////////
/////////////////////////////////////////////////////////////////////////////////////
/////////////////////////////////////////////////////////////////////////////////////
ET10_IrEtapa_1_ResetVacio_EnReposo:NOP   0;
      CLR;
      =     #Ir_PosicionReposo;
      =     #Ir_PosicionDescarga;

      L     1;
      T     #EstadoAsociadoEnMesa;
      JU    ETAPA_01_EnReposo;


NETWORK
TITLE = ETAPA 11 >>> RESET CARGADO >>> En Espera Descarga
/////////////////////////////////////////////////////////////////////////////////////
/////////////////////////////////////////////////////////////////////////////////////
// Extraer Destino
ETAPA_11_ResetCargado_EnEsperaDesCarga:NOP   0;
      SET;
      =     "DB900_Estado_Mesas".EstadoVI[#MesaDeDescarga].Etapas_Reset;


/////////////////////////////////////////////////////////////////////////////////////
// tenemos que comprobar si seguimos en la ventana, sino nos retiramos
      SET;
      AN    #pHs_Protrusion;
      JC    ErrorProtrusion;


/////////////////////////////////////////////////////////////////////////////////////
/////////////////////////////////////////////////////////////////////////////////////
/////////////////////////////////////////////////////////////////////////////////////
      SET;
      =     #PararElevador;
      CLR;
      =     #Ir_PosicionDescarga;
      =     #Ir_PosicionReposo;


/////////////////////////////////////////////////////////////////////////////////////
      SET;
      =     #NXT_AVTF;

      SET;
      A     #NXT_PTF;
      JC    ET11_IrEtapa_12_ResetCargado_EnDesCargaActiva;

      BE;


/////////////////////////////////////////////////////////////////////////////////////
/////////////////////////////////////////////////////////////////////////////////////
/////////////////////////////////////////////////////////////////////////////////////
ET11_IrEtapa_12_ResetCargado_EnDesCargaActiva:NOP   0;
      L     12;
      T     #EstadoAsociadoEnMesa;
      JU    ETAPA_12_ResetCargado_EnDescargaActiva;



NETWORK
TITLE = ETAPA 12 >>> RESET CARGADO >>> Descarga Activa
/////////////////////////////////////////////////////////////////////////////////////
/////////////////////////////////////////////////////////////////////////////////////
/////////////////////////////////////////////////////////////////////////////////////
// Proceso de descarga activa
// Tenemos que esperar a dejar de ver los dos detectores antes de dar por finalizado el proceso de descarga
ETAPA_12_ResetCargado_EnDescargaActiva:NOP   0;
      SET;
      =     "DB900_Estado_Mesas".EstadoVI[#MesaDeDescarga].Etapas_Descarga_S3;
      =     "DB900_Estado_Mesas".EstadoVI[#MesaDeDescarga].Etapas_Reset;


/////////////////////////////////////////////////////////////////////////////////////
      SET;
      =     #NXT_AVTF;
      =     #NXT_DescargaActiva;
      =     #PararElevador;

      SET;
      A     #NXT_PTF;
      =     #Avance_SalidaMovil;

      SET;
      AN    #FILTRO_PosicionDesCarga;
      A     #pHs_Protrusion;
      A     #NXT_FTF;
      JC    ET12_IrEtapa_13_ResetCargado_FinDescarga;

      BE;


/////////////////////////////////////////////////////////////////////////////////////
/////////////////////////////////////////////////////////////////////////////////////
/////////////////////////////////////////////////////////////////////////////////////
ET12_IrEtapa_13_ResetCargado_FinDescarga:NOP   0;
      CLR;
      =     #NXT_DescargaActiva;
      =     #NXT_AVTF;
      =     #ElevadorEnLenta;
      =     #Avance_SalidaMovil;

      L     13;
      T     #EstadoAsociadoEnMesa;
      JU    ETAPA_13_ResetCargado_FinDescarga;



NETWORK
TITLE = ETAPA 13 >>> RESET CARGADO >>> Fin Descarga
/////////////////////////////////////////////////////////////////////////////////////
/////////////////////////////////////////////////////////////////////////////////////
/////////////////////////////////////////////////////////////////////////////////////
ETAPA_13_ResetCargado_FinDescarga:NOP   0;
      SET;
      =     "DB900_Estado_Mesas".EstadoVI[#MesaDeDescarga].Etapas_Descarga_S3;
      =     "DB900_Estado_Mesas".EstadoVI[#MesaDeDescarga].Etapas_Reset;

/////////////////////////////////////////////////////////////////////////////////////
      SET;
      =     #PararElevador;

      CLR;
      =     #NXT_DescargaActiva;
      =     #NXT_AVTF;
      =     #ElevadorEnLenta;
      =     #Avance_SalidaMovil;


/////////////////////////////////////////////////////////////////////////////////////
/////////////////////////////////////////////////////////////////////////////////////
/////////////////////////////////////////////////////////////////////////////////////
      JU    ET13_FINAL_PasoDeDatos;


/////////////////////////////////////////////////////////////////////////////////////
/////////////////////////////////////////////////////////////////////////////////////
/////////////////////////////////////////////////////////////////////////////////////
ET13_FINAL_PasoDeDatos:NOP   0;
      L     7;
      T     #EstadoAsociadoEnMesa;
      JU    ETAPA_14_ResetCargado_MoverPosicionReposo;



NETWORK
TITLE = ETAPA 14 >>> RESET CARGADO >>> Mover a Posicion de Reposo
/////////////////////////////////////////////////////////////////////////////////////
/////////////////////////////////////////////////////////////////////////////////////
/////////////////////////////////////////////////////////////////////////////////////
// inicio del proceso de vuelta a reposo
ETAPA_14_ResetCargado_MoverPosicionReposo:NOP   0;
      SET;
      =     "DB900_Estado_Mesas".EstadoVI[#MesaDeDescarga].Etapas_Descarga_S3;
      =     "DB900_Estado_Mesas".EstadoVI[#MesaDeDescarga].Etapas_Reset;


/////////////////////////////////////////////////////////////////////////////////////
// tenemos que comprobar si seguimos en la ventana, sino nos retiramos
      SET;
      AN    #pHs_Protrusion;
      JC    ErrorProtrusion;


/////////////////////////////////////////////////////////////////////////////////////
/////////////////////////////////////////////////////////////////////////////////////
/////////////////////////////////////////////////////////////////////////////////////
      SET;
      A     #En_PosicionReposo;
      JC    ET14_IrEtapa_01_ResetCargado_EnReposo;

/////////////////////////////////////////////////////////////////////////////////////
      SET;
      =     #PararElevador;
      =     #Ir_PosicionReposo;

      CLR;
      =     #Ir_PosicionDescarga;

      BE;


/////////////////////////////////////////////////////////////////////////////////////
/////////////////////////////////////////////////////////////////////////////////////
/////////////////////////////////////////////////////////////////////////////////////
ET14_IrEtapa_01_ResetCargado_EnReposo:NOP   0;
      CLR;
      =     #Ir_PosicionReposo;
      =     #ElevadorEnLenta;

      L     1;
      T     #EstadoAsociadoEnMesa;
      JU    ETAPA_01_EnReposo;



NETWORK
TITLE = >>>>>>>>>>>>>>>>>>>>>>>>>>>>>>>>>>>>>>>>>>>>>>>>>>>>>>>>>>>>>>>>>>>

NETWORK
TITLE = ERRRORES DE LA MESA >>> Activacion
/////////////////////////////////////////////////////////////////////////////////////
/////////////////////////////////////////////////////////////////////////////////////
/////////////////////////////////////////////////////////////////////////////////////
ErrorProtrusion:SET;
      =     #PararElevador;
      =     "DB900_Estado_Mesas".EstadoVI[#MesaDeDescarga].Error_Mx;
      =     "DB900_Estado_Mesas".EstadoVI[#MesaDeDescarga].Err_Protusion;
      BE;

/////////////////////////////////////////////////////////////////////////////////////
/////////////////////////////////////////////////////////////////////////////////////
/////////////////////////////////////////////////////////////////////////////////////
ErrorMoverPosicionDescarga:SET;
      =     #PararElevador;
      =     "DB900_Estado_Mesas".EstadoVI[#MesaDeDescarga].Error_Mx;
      =     "DB900_Estado_Mesas".EstadoVI[#MesaDeDescarga].Err_Tout_Sacar;
      BE;

/////////////////////////////////////////////////////////////////////////////////////
/////////////////////////////////////////////////////////////////////////////////////
/////////////////////////////////////////////////////////////////////////////////////
ErrorMoverPosicionReposo:SET;
      =     #PararElevador;
      =     "DB900_Estado_Mesas".EstadoVI[#MesaDeDescarga].Error_Mx;
      =     "DB900_Estado_Mesas".EstadoVI[#MesaDeDescarga].Err_Tout_Recoger;
      BE;

/////////////////////////////////////////////////////////////////////////////////////
/////////////////////////////////////////////////////////////////////////////////////
/////////////////////////////////////////////////////////////////////////////////////
ErrorPerdidaPresencia:NOP   0;  // error de Perdida de Presencia
      SET;
      =     "DB900_Estado_Mesas".EstadoVI[#MesaDeDescarga].Error_Mx;
      =     "DB900_Estado_Mesas".EstadoVI[#MesaDeDescarga].Err_Perdida_PHs;
      =     #PararElevador;
      BE;

/////////////////////////////////////////////////////////////////////////////////////
/////////////////////////////////////////////////////////////////////////////////////
/////////////////////////////////////////////////////////////////////////////////////
ErrorDatosCargada:NOP   0;  // error en la carga
      SET;
      =     "DB900_Estado_Mesas".EstadoVI[#MesaDeDescarga].Error_Mx;
      =     "DB900_Estado_Mesas".EstadoVI[#MesaDeDescarga].Err_DatosPLC;
      =     #PararElevador;
      BE;



NETWORK
TITLE = FIN DE LA FUNCION
/////////////////////////////////////////////////////////////////////////////////////
/////////////////////////////////////////////////////////////////////////////////////
/////////////////////////////////////////////////////////////////////////////////////
FinFuncion:BE;


END_FUNCTION_BLOCK
